PROGRAM MAIN_1
VAR
	(* Visu Elements*)
	sLine1				:STRING := 'Hello';
	sLine2				:STRING := 'Beckhoff';

	(* Linked Varaibles *)
	SlavePort  AT %I* 	: WORD;
	SlaveNetID AT %I* 	: T_AmsNetIdArr;

	fbTrig				: R_TRIG;
	M_1					: BOOL;
	fb_EL6090			: FB_EL6090;

	StrTime				: ST_OperatingTime;

	EL6090_State AT %I*	: WORD;
END_VAR

IF EL6090_State=16#8 THEN
	fb_EL6090.bAutoUpdate:=TRUE;
END_IF


fb_EL6090(bAutoUpdate:=,
		AmsNetId:=F_CreateAmsNetId(SlaveNetId),
		Port:=SlavePort);
StrTime:=f_Convert_to_OperatingTime(fb_EL6090.nOpertingTime);


(* pos. trig from NAVI "ENTER"*)
fbTrig(CLK:=GVL_CouplerOnDesk.bNavEnter);
IF fbTrig.Q THEN
	M_1:=NOT M_1;
	GVL_CouplerOnDesk.nDisplayRow1:=GVL_CouplerOnDesk.nDisplayRow1+1;
END_IF

GVL_CouplerOnDesk.nDisplayRow2:=GVL_CouplerOnDesk.nDisplayRow2+1;

IF M_1 THEN
	fb_EL6090.strLine_1:=sLine1;
	fb_EL6090.strLine_2:=sLine2;
ELSE
	fb_EL6090.strLine_1:='Value 1:%i';
	fb_EL6090.strLine_2:='Value 2:%i';
END_IF

END_PROGRAM

(* stored: Version 1.1.0.1
   POU MAIN_1: Id {f999584f-bbe1-4811-b1b2-84f8b34e0f17}, SpecialFunc None *)
